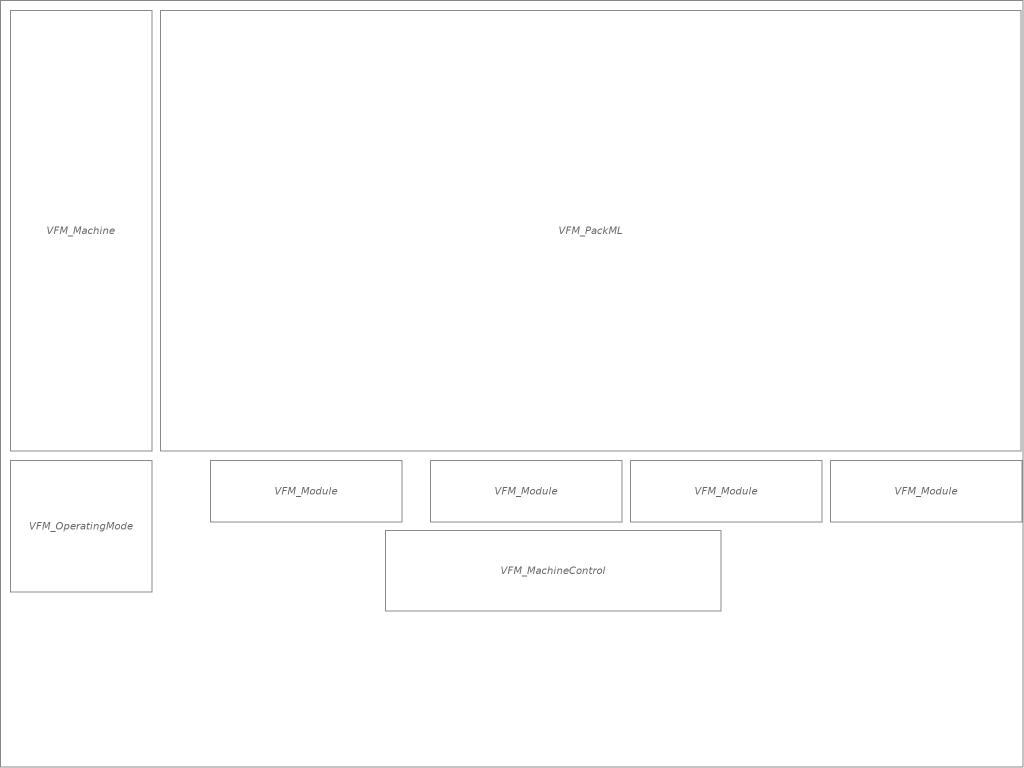
VISUALIZATION VIS_Main  // 1024x768
    Frame (160,10 861x441)
        shows VFM_PackML(HMI := MAIN.Machine.PackMLBaseModule_HMI)
    Frame (385,530 336x81)
        shows VFM_MachineControl(HMI := MAIN.Machine.HMI)
    Frame (10,10 142x441)
        shows VFM_Machine(HMI := MAIN.Machine.PackMLBaseModule_HMI)
    Frame (10,460 142x132)
        shows VFM_OperatingMode(HMI := MAIN.Machine.PackMLBaseModule_HMI)
    Frame (210,460 192x62)
        shows VFM_Module(HMI := MAIN.Machine.PackMLBaseModule_HMI)
    Frame (430,460 192x62)
        shows VFM_Module(HMI := MAIN.Machine.EM_Infeed.PackMLBaseModule_HMI)
    Frame (630,460 192x62)
        shows VFM_Module(HMI := MAIN.Machine.EM_Work.PackMLBaseModule_HMI)
    Frame (830,460 192x62)
        shows VFM_Module(HMI := MAIN.Machine.EM_Outfeed.PackMLBaseModule_HMI)
END_VISUALIZATION

(* stored: Version 1.1.0.1, ProductVersion 3.1.4024.12
   Visu VIS_Main: Id {4fef3d91-e7d6-44a9-99cf-6c06f81453b1} *)
